INTERFACE ITcoContext EXTENDS ITcoObject

PROPERTY EndCycleCount : ULINT
GET
END_GET
END_PROPERTY

PROPERTY Environment : ITcoContextEnvironment
GET
END_GET
END_PROPERTY

PROPERTY RealTimeClock : ITcoRtc
GET
END_GET
END_PROPERTY

PROPERTY StartCycleCount : ULINT
GET
END_GET
END_PROPERTY

END_INTERFACE

(* stored: Version 1.1.0.1, ProductVersion 3.1.4024.9
   Itf ITcoContext: Id {403f0fe8-301c-472b-9683-fcc2c906813c}
   Property EndCycleCount: Id {0ef1070c-3626-47f3-b7ff-b49194a10cb0}
   Get Get: Id {178bc67c-e591-409d-b72b-c8116e29fd92}
   Property Environment: Id {6eaa7498-1d19-0a13-0e89-7e25c3e22943}
   Get Get: Id {29de8b00-48da-0196-233a-df201ec80325}
   Property RealTimeClock: Id {a8f4d1c6-2d8d-0ba5-21b5-6c50c789cfac}
   Get Get: Id {687aebad-3b3d-04fd-11f3-3dbbbbe35dfb}
   Property StartCycleCount: Id {07375695-36dd-4eef-96de-a19ffb2e7fb5}
   Get Get: Id {777fb9d8-cfe2-4a4e-8b02-06212d36a736} *)
